    PROC rWireCut()
        VAR jointtarget jTepmCut{10};
        VAR speeddata vTempFast;
        VAR speeddata vTempSlow;
        vTempFast:=[nWireCutSpeed,500,nWireCutSpeed,100];
        vTempSlow:=[nWireCutSpeed/3,500,nWireCutSpeed/3,100];
        PulseDO\PLength:=nInchingTime,soAwManFeedFwd;
        Reset do09_Wire_Cutter_Close;
        Set do10_Wire_Cutter_Open;
        !      WaitTime 2.25;
        jWireCut4.robax:=[90,90,-50,0,0,0];
        MoveAbsJ jWireCut4\NoEOffs,vTempFast,z100,tWeld1;
        MoveAbsJ jWireCut3\NoEOffs,vTempFast,z100,tWeld1;
        MoveAbsJ jWireCut2\NoEOffs,vTempFast,z100,tWeld1;
        MoveAbsJ jWireCut1\NoEOffs,vTempFast,z10,tWeld1;
        WaitRob\ZeroSpeed;
        WaitTime 0.3;
        MoveAbsJ jWireCut0\NoEOffs,vTempSlow,z0,tWeld1;
        IF bWireCutSync=TRUE WaitSyncTask Wait{90},taskGroup12;
        WaitRob\ZeroSpeed;
        WaitTime 0.5;
        Reset do10_Wire_Cutter_Open;
        PulseDO\PLength:=1,do09_Wire_Cutter_Close;
        WaitTime 0.5;
        PulseDO\PLength:=1,do10_Wire_Cutter_Open;
        WaitTime 1;
        MoveAbsJ jWireCut1\NoEOffs,vTempSlow,z100,tWeld1;
        WaitRob\ZeroSpeed;
        MoveAbsJ jWireCut2\NoEOffs,vTempFast,z100,tWeld1;
        MoveAbsJ jWireCut3\NoEOffs,vTempFast,z100,tWeld1;
        MoveAbsJ jWireCut4\NoEOffs,vTempFast,z100,tWeld1;
        WaitRob\ZeroSpeed;
        Reset do10_Wire_Cutter_Open;
        stReact{1}:="WireCutOk";
        WaitUntil stCommand="";
        stReact{1}:="Ready";
        WaitUntil stReact=["Ready","Ready","Ready"];
        RETURN ;
    ENDPROC

    PROC rWireCutMove()
        VAR jointtarget jTepmCut{10};
        VAR speeddata vTempFast;
        VAR speeddata vTempSlow;
        vTempFast:=[nWireCutSpeed,500,nWireCutSpeed,100];
        vTempSlow:=[nWireCutSpeed/3,500,nWireCutSpeed/3,100];
        PulseDO\PLength:=nInchingTime,soAwManFeedFwd;
        Reset do09_Wire_Cutter_Close;
        Set do10_Wire_Cutter_Open;
        !      WaitTime 2.25;
        MoveAbsJ jWireCut3\NoEOffs,vTempFast,z100,tWeld1;
        MoveAbsJ jWireCut2\NoEOffs,vTempFast,z100,tWeld1;
        MoveAbsJ jWireCut1\NoEOffs,vTempFast,z10,tWeld1;
        WaitRob\ZeroSpeed;
        WaitTime 0.3;
        MoveAbsJ jWireCut0\NoEOffs,vTempSlow,z0,tWeld1;
        IF bWireCutSync=TRUE WaitSyncTask Wait{90},taskGroup12;
        WaitRob\ZeroSpeed;
        WaitTime 0.5;
        Reset do10_Wire_Cutter_Open;
        PulseDO\PLength:=1,do09_Wire_Cutter_Close;
        WaitTime 0.5;
        PulseDO\PLength:=1,do10_Wire_Cutter_Open;
        WaitTime 1;
        MoveAbsJ jWireCut1\NoEOffs,vTempSlow,z100,tWeld1;
        WaitRob\ZeroSpeed;
        MoveAbsJ jWireCut2\NoEOffs,vTempFast,z100,tWeld1;
        IF bWirecut=[FALSE,TRUE,FALSE] THEN
            MoveAbsJ jWireCut3\NoEOffs,vTempFast,z100,tWeld1;
            jWireCut4.robax:=[40,90,-90,0,0,0];
            MoveAbsJ jWireCut4\NoEOffs,vTempFast,z100,tWeld1;
        ENDIF
        WaitRob\ZeroSpeed;
        Reset do10_Wire_Cutter_Open;
        stReact{1}:="WireCutOk";
        WaitUntil stCommand="";
        stReact{1}:="Ready";
        WaitUntil stReact=["Ready","Ready","Ready"];
        RETURN ;
    ENDPROC

    PROC rWireCutShot()
        VAR jointtarget jTepmCut{10};
        VAR speeddata vTempFast;
        VAR speeddata vTempSlow;
        vTempFast:=[nWireCutSpeed,500,nWireCutSpeed,100];
        vTempSlow:=[nWireCutSpeed/3,500,nWireCutSpeed/3,100];
        PulseDO\PLength:=nInchingTime,soAwManFeedFwd;
        Reset do09_Wire_Cutter_Close;
        Set do10_Wire_Cutter_Open;
        WaitTime nInchingTime;
        MoveAbsJ jWireCut1\NoEOffs,vTempFast,z10,tWeld1;
        WaitRob\ZeroSpeed;
        WaitTime 0.3;
        MoveAbsJ jWireCut0\NoEOffs,vTempSlow,z0,tWeld1;
        IF bWireCutSync=TRUE WaitSyncTask Wait{90},taskGroup12;
        WaitRob\ZeroSpeed;
        WaitTime 0.5;
        Reset do10_Wire_Cutter_Open;
        PulseDO\PLength:=1,do09_Wire_Cutter_Close;
        WaitTime 0.5;
        PulseDO\PLength:=1,do10_Wire_Cutter_Open;
        WaitTime 1;
        MoveAbsJ jWireCut1\NoEOffs,vTempSlow,z100,tWeld1;
        WaitRob\ZeroSpeed;
        MoveAbsJ jWireCut2\NoEOffs,vTempFast,z100,tWeld1;
        WaitRob\ZeroSpeed;
        Reset do10_Wire_Cutter_Open;
        stReact{1}:="WireCutOk";
        WaitUntil stCommand="";
        stReact{1}:="Ready";
        WaitUntil stReact=["Ready","Ready","Ready"];
        RETURN ;
    ENDPROC

    PROC rTrapNoWeldMove()
        VAR num i;
        VAR targetdata WeldsTemp;
        VAR robtarget pWeldTemp;
        VAR num nTempMmps;
        VAR speeddata vWeldTemp;
        IDelete inumMoveG_PosHold;
        StopMove;
        !        ClearPath;
        !        StorePath;

        i:=nRunningStep{1};
        nTempMmps:=Welds1{i}.cpm/6;
        vWeldTemp:=[nTempMmps,200,200,200];

        pWeldTemp:=CRobT(\taskname:="T_ROB1"\Tool:=tWeld1\WObj:=wobjWeldLine1);
        StartMove;
        ConfL\Off;
        WHILE (so_MoveG_PosHold=1) DO
            nTrapCheck_1:=2;
            MoveL Offs(pWeldTemp,0,0,0),vWeldTemp,fine,tWeld1\WObj:=wobjWeldLine1;
            MoveL Offs(pWeldTemp,0,0,0),vWeldTemp,fine,tWeld1\WObj:=wobjWeldLine1;
        ENDWHILE
        ConfL\On;
        !        RestoPath;
    ENDPROC

    PROC rCorrSearchStartEnd()
        VAR num TempHeight;
        VAR num TempBreadth;
        VAR num Temp_X;
        VAR num Temp_Y;
        VAR num nHeightBuffer;
        VAR num n_X;
        VAR num n_Y;
        VAR num n_Z;
        VAR num n_Ret_X;
        VAR num n_Ret_Y;
        VAR num n_Ret_Z;
        VAR robtarget pTemp;
        VAR robtarget pCorrTemp_Start{2};
        VAR jointtarget jCorrTemp_Start{2};
        VAR robtarget pCorrTemp_End{2};
        VAR jointtarget jCorrTemp_End{2};

        RetryDepthData:=[10,10,10];
        IDelete iErrorDuringEntry;
        CONNECT iErrorDuringEntry WITH trapErrorDuringEntry;
        ISignalDO intTouch_1,1,iErrorDuringEntry;
        ISleep iErrorDuringEntry;

        bInstalldir:=bRobSwap;
        IF bRobSwap=FALSE THEN
            edgestartBuffer1:=edgeStart{1};
            edgeEndBuffer1:=edgeEnd{1};
        ELSE
            edgestartBuffer1:=edgeStart{2};
            edgeEndBuffer1:=edgeEnd{2};
        ENDIF
        WaitRob\ZeroSpeed;
        WaitSyncTask Wait{20},taskGroup123;

        WaitUntil bGanTry_Last_pos=TRUE;
        !        IF pi29_NextCmd=1 nTouchRetryCount{1}:=0;

        nCorrFailOffs_Z:=10*nEntryRetryCount{1};
        IF bRobSwap=TRUE nCorrFailOffs_Y:=(10*nEntryRetryCount{1});
        IF bRobSwap=FALSE nCorrFailOffs_Y:=(10*nEntryRetryCount{1});


        TEST nMacro001{1}
        CASE 0,1,2,3,4,5,8:
            IF edgeEndBuffer1.Breadth<edgeEndBuffer1.Height THEN
                ! Setting Conditions
                IF nMacro001{1}=0 OR nMacro001{1}=1 OR nMacro001{1}=2 OR nMacro001{1}=5 n_X:=-15;
                IF nMacro001{1}=3 OR nMacro001{1}=4 OR nMacro001{1}=8 n_X:=0;
                !                n_Y:=TouchLimit(corrEnd{nMacro001{1}+1}.Y_StartOffset+nEndThick,edgeEndBuffer1.Breadth)+nCorrFailOffs_Y;
                n_Y:=corrEnd{nMacro001{1}+1}.Y_StartOffset+nEndThick+nCorrFailOffs_Y;
                n_Ret_Y:=TouchLimit(corrEnd{nMacro001{1}+1}.Y_ReturnLength,edgeEndBuffer1.Breadth);
                n_Ret_Z:=TouchLimit(corrEnd{nMacro001{1}+1}.Z_ReturnLength,edgeEndBuffer1.Height);
                n_Z:=TouchLimit(corrEnd{nMacro001{1}+1}.Z_StartOffset,edgeEndBuffer1.Height)+nCorrFailOffs_Z;

                ! Touch Entry Location================================================================
                IWatch iErrorDuringEntry;

                rCheckWelder;

                rMoveCorrConnect n_X,n_Y,n_Z,0,0,0,nHeightBuffer,bEnd,bInstalldir\LIN;
                Reset soLn1Touch;
                IDelete iErrorDuringEntry;

                !                IF bTouchWorkCount{3}=TRUE GOTO TouchComplete_End_Y;
                WaitTime 0;
                !                 rCheckTouchAtStart;
                !=====================================================================================
                ! edge_Y
                IF bTouchWorkCount{1}=FALSE THEN
                    rCorrSearchWeldLineEdgeY n_X,n_Y,n_Z,corrEnd{nMacro001{1}+1}.Y_Depth+nCorrFailOffs_Y+nEndThick,n_Ret_Y,bEnd,bInstalldir,"End_Y";
                    bTouchWorkCount{1}:=TRUE;
                    nTouchRetryCount{1}:=0;
                ENDIF

                ! edge_Z
                IF bTouchWorkCount{2}=FALSE THEN
                    !                 Setting Conditions
                    n_Y:=n_Ret_Y;
                    n_Ret_Z:=TouchLimit(corrEnd{nMacro001{1}+1}.Z_ReturnLength,edgeEndBuffer1.Height);

                    rCorrSearchWeldLineEdgeZ n_X,n_Y,n_Z,corrEnd{nMacro001{1}+1}.Z_Depth+nCorrFailOffs_Z,n_Ret_Z,bEnd,bInstalldir,"End_Z";
                    bTouchWorkCount{2}:=TRUE;
                    nTouchRetryCount{1}:=0;
                ENDIF

                ! Setting Conditions
                n_Z:=n_Ret_Z;
                rMoveCorrConnect n_X,n_Y,n_Z,0,0,0,nHeightBuffer,bEnd,bInstalldir;

                IF nMacro001{1}=3 OR nMacro001{1}=4 OR nMacro001{1}=8 GOTO TouchComplete_End_Y;
                IF nMacro001{1}=2 OR nMacro001{1}=5 THEN
                    IF nMacro001{1}=5 n_Z:=edgeEndBuffer1.HoleSize+1;
                ELSE
                    ! Setting Conditions
                    n_X:=corrEnd{nMacro001{1}+1}.X_StartOffset;
                    rMoveCorrConnect n_X,n_Y,n_Z,0,0,0,nHeightBuffer,bEnd,bInstalldir;
                    ! Setting Conditions
                    n_Y:=-5;
                    rMoveCorrConnect n_X,n_Y,n_Z,0,0,0,nHeightBuffer,bEnd,bInstalldir;

                ENDIF

                ! edge_X
                IF bTouchWorkCount{3}=FALSE THEN
                    rCorrSearchWeldLineEdgeX n_X,n_Y,n_Z,corrEnd{nMacro001{1}+1}.X_Depth,corrEnd{nMacro001{1}+1}.X_ReturnLength,bEnd,bInstalldir,"End_X";
                    bTouchWorkCount{3}:=TRUE;
                    nTouchRetryCount{1}:=0;
                ENDIF
                ! Setting Conditions
                n_X:=corrEnd{nMacro001{1}+1}.X_ReturnLength;
                rMoveCorrConnect n_X,n_Y,n_Z,0,corrEnd{nMacro001{1}+1}.RY_Torch,0,nHeightBuffer,bEnd,bInstalldir;
                ! Labal
                TouchComplete_End_Y:
                ! Setting Conditions
                n_Y:=n_Ret_Y;
                rMoveCorrConnect n_X,n_Y,n_Z,0,corrEnd{nMacro001{1}+1}.RY_Torch+n_Angle,0,nHeightBuffer,bEnd,bInstalldir;

            ELSE

                ! Setting Conditions
                IF nMacro001{1}=0 OR nMacro001{1}=1 OR nMacro001{1}=2 OR nMacro001{1}=5 n_X:=-15;
                IF nMacro001{1}=3 OR nMacro001{1}=4 OR nMacro001{1}=8 n_X:=0;
                n_Y:=TouchLimit(corrEnd{nMacro001{1}+1}.Y_StartOffset+nEndThick,edgeEndBuffer1.Breadth)+nCorrFailOffs_Y;
                n_Ret_Y:=TouchLimit(corrEnd{nMacro001{1}+1}.Y_ReturnLength,edgeEndBuffer1.Breadth);
                n_Ret_Z:=TouchLimit(corrEnd{nMacro001{1}+1}.Z_ReturnLength,edgeEndBuffer1.Height);
                n_Z:=TouchLimit(corrEnd{nMacro001{1}+1}.Z_StartOffset,edgeEndBuffer1.Height)+nCorrFailOffs_Z;

                IWatch iErrorDuringEntry;

                rCheckWelder;

                rMoveCorrConnect n_X,n_Y,n_Z,0,0,0,nHeightBuffer,bEnd,bInstalldir\LIN;
                Reset soLn1Touch;
                IDelete iErrorDuringEntry;

                !                IF bTouchWorkCount{3}=TRUE GOTO TouchComplete_End_Z;
                WaitTime 0;
                !    rCheckTouchAtStart;

                ! edge_Z
                IF bTouchWorkCount{1}=FALSE THEN
                    rCorrSearchWeldLineEdgeZ n_X,n_Y,n_Z,corrEnd{nMacro001{1}+1}.Z_Depth+nCorrFailOffs_Z,n_Ret_Z,bEnd,bInstalldir,"End_Z";
                    bTouchWorkCount{1}:=TRUE;
                    nTouchRetryCount{1}:=0;
                ENDIF

                ! edge_Y
                IF bTouchWorkCount{2}=FALSE THEN
                    ! Setting Conditions
                    n_Ret_Y:=TouchLimit(corrEnd{nMacro001{1}+1}.Y_ReturnLength,edgeEndBuffer1.Breadth);
                    n_Z:=n_Ret_Z;
                    rCorrSearchWeldLineEdgeY n_X,n_Y,n_Z,corrEnd{nMacro001{1}+1}.Y_Depth+nCorrFailOffs_Y+nEndThick,n_Ret_Y,bEnd,bInstalldir,"End_Y";
                    bTouchWorkCount{2}:=TRUE;
                    nTouchRetryCount{1}:=0;
                ENDIF

                ! Setting Conditions
                n_Y:=n_Ret_Y;
                rMoveCorrConnect n_X,n_Y,n_Z,0,0,0,nHeightBuffer,bEnd,bInstalldir;

                IF nMacro001{1}=3 OR nMacro001{1}=4 OR nMacro001{1}=8 GOTO TouchComplete_End_Z;
                IF nMacro001{1}=2 OR nMacro001{1}=5 THEN
                    IF nMacro001{1}=5 n_Z:=edgeEndBuffer1.HoleSize+1;
                ELSE

                    ! Setting Conditions
                    n_X:=corrEnd{nMacro001{1}+1}.X_StartOffset;
                    rMoveCorrConnect n_X,n_Y,n_Z,0,0,0,nHeightBuffer,bEnd,bInstalldir;
                    ! Setting Conditions
                    n_Y:=-5;
                    rMoveCorrConnect n_X,n_Y,n_Z,0,0,0,nHeightBuffer,bEnd,bInstalldir;

                ENDIF

                ! edge_X
                IF bTouchWorkCount{3}=FALSE THEN
                    rCorrSearchWeldLineEdgeX n_X,n_Y,n_Z,corrEnd{nMacro001{1}+1}.X_Depth,corrEnd{nMacro001{1}+1}.X_ReturnLength,bEnd,bInstalldir,"End_X";
                    bTouchWorkCount{3}:=TRUE;
                    nTouchRetryCount{1}:=0;
                ENDIF

                ! Setting Conditions
                n_X:=corrEnd{nMacro001{1}+1}.X_ReturnLength;
                rMoveCorrConnect n_X,n_Y,n_Z,0,corrEnd{nMacro001{1}+1}.RY_Torch,0,nHeightBuffer,bEnd,bInstalldir;
                ! Labal
                TouchComplete_End_Z:
                ! Setting Conditions
                n_Y:=n_Ret_Y;
                rMoveCorrConnect n_X,n_Y,n_Z,0,corrEnd{nMacro001{1}+1}.RY_Torch+n_Angle,0,nHeightBuffer,bEnd,bInstalldir;
            ENDIF
            IF nMacro001{1}=3 OR nMacro001{1}=4 OR nMacro001{1}=8 THEN
                !   IF bEndSearchComplete=FALSE pCorredSplitPos:=ConvertPosWeldLineToFloor(pSearchStart,nWeldLineLength+nCorrX_Store_End,nCorrY_Store_End,nCorrZ_Store_End);
            ENDIF
        CASE 9:
            !   pCorredEndPos:=pCorredSplitPos;
        DEFAULT:
            Stop;
            Stop;
            ExitCycle;
        ENDTEST

        !        IF abs(pCheckBuffer{2}.trans.x-pCheckBuffer{3}.trans.x)<5 rTouchErrorHandling 13;
        !        IF abs(pCheckBuffer{2}.trans.Y-pCheckBuffer{3}.trans.Y)<5 rTouchErrorHandling 13;
        !        IF abs(pCheckBuffer{2}.trans.Z-pCheckBuffer{3}.trans.Z)<5 rTouchErrorHandling 13;

        bTouch_last_R1_Comp:=TRUE;
        bTouch_First_R1_Comp:=FALSE;
        pCorrTemp_End{1}:=CRobT(\TaskName:="T_ROB1"\Tool:=tWeld1\WObj:=wobjWeldLine1);
        pCorrTemp_End{1}.trans:=[nWeldLineLength_R1+nCorrX_Store_End{1},nCorrY_Store_End{1},nCorrZ_Store_End{1}];
        jCorrTemp_End{1}:=CalcJointT(pCorrTemp_End{1},tWeld1\WObj:=wobjWeldLine1);
        pCorrT_ROB1_End:=CalcRobT(jCorrTemp_End{1},Tool:=tWeld1\WObj:=wobjRotCtr1);
        WaitUntil bGanTry_First_pos=TRUE AND bTouch_last_R2_Comp=TRUE;

        !!! Start correctioning from start edge !!!
        TEST nMacro010{1}
        CASE 0,1,2,3,4,5:
            IF edgestartBuffer1.Breadth<edgestartBuffer1.Height THEN

                ! Setting Conditions
                IF nMacro010{1}=0 OR nMacro010{1}=1 OR nMacro010{1}=2 OR nMacro010{1}=5 n_X:=-15;
                IF nMacro010{1}=3 OR nMacro010{1}=4 OR nMacro010{1}=8 n_X:=0;
                !                n_Y:=TouchLimit(corrStart{nMacro010{1}+1}.Y_StartOffset+nStartThick,edgeStartBuffer1.Breadth)+nCorrFailOffs_Y;
                n_Y:=corrStart{nMacro010{1}+1}.Y_StartOffset+nStartThick+nCorrFailOffs_Y;
                n_Ret_Y:=TouchLimit(corrStart{nMacro010{1}+1}.Y_ReturnLength,edgestartBuffer1.Breadth);
                n_Z:=TouchLimit(corrStart{nMacro010{1}+1}.Z_StartOffset,edgestartBuffer1.Height)+nCorrFailOffs_Z;
                n_Ret_Z:=TouchLimit(corrStart{nMacro010{1}+1}.Z_ReturnLength,edgestartBuffer1.Height);

                ! edge_Y
                rMoveCorrConnect n_X,n_Y,n_Z,0,corrStart{nMacro010{1}+1}.RY_Torch+n_Angle,0,nHeightBuffer,bStart,bInstalldir\LIN;
                !    rCheckTouchAtStart;

                IF bTouchWorkCount{4}=FALSE THEN
                    rCorrSearchWeldLineEdgeY n_X,n_Y,n_Z,corrStart{nMacro010{1}+1}.Y_Depth+nCorrFailOffs_Y+nStartThick,n_Ret_Y,bStart,bInstalldir,"Start_Y";
                    bTouchWorkCount{4}:=TRUE;
                    nTouchRetryCount{1}:=0;
                ENDIF

                ! edge_Z
                IF bTouchWorkCount{5}=FALSE THEN
                    ! Setting Conditions
                    n_Y:=n_Ret_Y;
                    n_Ret_Z:=TouchLimit(corrStart{nMacro010{1}+1}.Z_ReturnLength,edgestartBuffer1.Height);
                    rCorrSearchWeldLineEdgeZ n_X,n_Y,n_Z,corrStart{nMacro010{1}+1}.Z_Depth+nCorrFailOffs_Z,n_Ret_Z,bStart,bInstalldir,"Start_Z";
                    bTouchWorkCount{5}:=TRUE;
                    nTouchRetryCount{1}:=0;
                ENDIF

                ! Setting Conditions
                n_Z:=n_Ret_Z;
                rMoveCorrConnect n_X,n_Y,n_Z,0,0,0,nHeightBuffer,bStart,bInstalldir;

                IF nMacro010{1}=3 OR nMacro010{1}=4 OR nMacro010{1}=8 GOTO TouchComplete_Start_Y;
                IF nMacro010{1}=2 OR nMacro010{1}=5 THEN
                    IF nMacro010{1}=5 n_Z:=edgestartBuffer1.HoleSize+1;
                ELSE

                    ! Setting Conditions
                    n_X:=corrStart{nMacro010{1}+1}.X_StartOffset;
                    rMoveCorrConnect n_X,n_Y,n_Z,0,0,0,nHeightBuffer,bStart,bInstalldir;
                    ! Setting Conditions
                    n_Y:=-5;
                    rMoveCorrConnect n_X,n_Y,n_Z,0,0,0,nHeightBuffer,bStart,bInstalldir;
                ENDIF
                !    ENDIF

                ! edge_X
                IF bTouchWorkCount{6}=FALSE THEN
                    rCorrSearchWeldLineEdgeX n_X,n_Y,n_Z,corrStart{nMacro010{1}+1}.X_Depth,corrStart{nMacro010{1}+1}.X_ReturnLength,bStart,bInstalldir,"Start_X";
                    bTouchWorkCount{6}:=TRUE;
                    nTouchRetryCount{1}:=0;
                ENDIF
                ! Setting Conditions
                n_X:=corrStart{nMacro010{1}+1}.X_ReturnLength;
                rMoveCorrConnect n_X,n_Y,n_Z,0,corrStart{nMacro010{1}+1}.RY_Torch,0,nHeightBuffer,bStart,bInstalldir;
                ! Labal
                TouchComplete_Start_Y:
            ELSE

                ! Setting Conditions
                IF nMacro010{1}=0 OR nMacro010{1}=1 OR nMacro010{1}=2 OR nMacro010{1}=5 n_X:=-15;
                IF nMacro010{1}=3 OR nMacro010{1}=4 OR nMacro010{1}=8 n_X:=0;
                n_Y:=TouchLimit(corrStart{nMacro010{1}+1}.Y_StartOffset+nStartThick,edgestartBuffer1.Breadth)+nCorrFailOffs_Y;
                n_Ret_Y:=TouchLimit(corrStart{nMacro010{1}+1}.Y_ReturnLength,edgestartBuffer1.Breadth);
                n_Ret_Z:=TouchLimit(corrStart{nMacro010{1}+1}.Z_ReturnLength,edgestartBuffer1.Height);
                n_Z:=TouchLimit(corrStart{nMacro010{1}+1}.Z_StartOffset,edgestartBuffer1.Height)+nCorrFailOffs_Z;

                rMoveCorrConnect n_X,n_Y,n_Z,0,corrStart{nMacro010{1}+1}.RY_Torch+n_Angle,0,nHeightBuffer,bStart,bInstalldir\LIN;
                ! rCheckTouchAtStart;


                ! edge_Z
                IF bTouchWorkCount{4}=FALSE THEN
                    rCorrSearchWeldLineEdgeZ n_X,n_Y,n_Z,corrStart{nMacro010{1}+1}.Z_Depth+nCorrFailOffs_Z,n_Ret_Z,bStart,bInstalldir,"Start_Z";
                    bTouchWorkCount{4}:=TRUE;
                    nTouchRetryCount{1}:=0;
                ENDIF
                ! Setting Conditions


                ! edge_Y
                IF bTouchWorkCount{5}=FALSE THEN
                    ! Setting Conditions
                    n_Ret_Y:=TouchLimit(corrStart{nMacro010{1}+1}.Y_ReturnLength,edgestartBuffer1.Breadth);
                    n_Z:=n_Ret_Z;
                    rCorrSearchWeldLineEdgeY n_X,n_Y,n_Z,corrStart{nMacro010{1}+1}.Y_Depth+nCorrFailOffs_Y+nStartThick,n_Ret_Y,bStart,bInstalldir,"Start_Y";
                    bTouchWorkCount{5}:=TRUE;
                    nTouchRetryCount{1}:=0;
                ENDIF

                ! Setting Conditions
                n_Y:=n_Ret_Y;
                rMoveCorrConnect n_X,n_Y,n_Z,0,0,0,nHeightBuffer,bStart,bInstalldir;

                IF nMacro010{1}=3 OR nMacro010{1}=4 OR nMacro010{1}=8 GOTO TouchComplete_Start_Z;
                IF nMacro010{1}=2 OR nMacro010{1}=5 THEN
                    IF nMacro010{1}=5 n_Z:=edgestartBuffer1.HoleSize+1;
                ELSE
                    !    IF bTouchWorkCount{6}=FALSE THEN
                    ! Setting Conditions
                    n_X:=corrStart{nMacro010{1}+1}.X_StartOffset;
                    rMoveCorrConnect n_X,n_Y,n_Z,0,0,0,nHeightBuffer,bStart,bInstalldir;
                    ! Setting Conditions
                    n_Y:=-5;
                    rMoveCorrConnect n_X,n_Y,n_Z,0,0,0,nHeightBuffer,bStart,bInstalldir;
                ENDIF
                ! ENDIF

                ! edge_X
                IF bTouchWorkCount{6}=FALSE THEN
                    rCorrSearchWeldLineEdgeX n_X,n_Y,n_Z,corrStart{nMacro010{1}+1}.X_Depth,corrStart{nMacro010{1}+1}.X_ReturnLength,bStart,bInstalldir,"Start_X";
                    bTouchWorkCount{6}:=TRUE;
                    nTouchRetryCount{1}:=0;
                ENDIF
                ! Setting Conditions
                n_X:=corrStart{nMacro010{1}+1}.X_ReturnLength;
                rMoveCorrConnect n_X,n_Y,n_Z,0,corrStart{nMacro010{1}+1}.RY_Torch,0,nHeightBuffer,bStart,bInstalldir;

                ! Labal
                TouchComplete_Start_Z:
            ENDIF

        DEFAULT:
            Stop;
            Stop;
            ExitCycle;
        ENDTEST

        pTemp:=CRobT(\TaskName:="T_ROB1"\Tool:=tWeld1\WObj:=wobjWeldLine1);
        WaitRob\ZeroSpeed;
        MoveL RelTool(pTemp,0,0,-15),vTargetSpeed,zTargetZone,tWeld1\WObj:=wobjWeldLine1;

        bTouch_First_R1_Comp:=TRUE;
        bTouch_last_R1_Comp:=TRUE;

        WaitUntil bTouch_First_R2_Comp=TRUE;

        pCorrTemp_Start{1}:=CRobT(\TaskName:="T_ROB1"\Tool:=tWeld1\WObj:=wobjWeldLine1);
        pCorrTemp_Start{1}.trans:=[nCorrX_Store_Start{1},nCorrY_Store_Start{1},nCorrZ_Store_Start{1}];
        jCorrTemp_Start{1}:=CalcJointT(pCorrTemp_Start{1},tWeld1\WObj:=wobjWeldLine1);
        pCorrT_ROB1_Start:=CalcRobT(jCorrTemp_Start{1},Tool:=tWeld1\WObj:=wobjRotCtr1);








        stReact{1}:="CorrSearchOK";
        WaitUntil stCommand="";
        stReact{1}:="Ready";
        nCorrFailOffs_Y:=0;
        nCorrFailOffs_Z:=0;
        nCorrX_Store_Start{1}:=0;
        nCorrY_Store_Start{1}:=0;
        nCorrZ_Store_Start{1}:=0;
        nCorrX_Store_End{1}:=0;
        nCorrY_Store_End{1}:=0;
        nCorrZ_Store_End{1}:=0;
    ENDPROC

    PROC rMoveCorrConnect(num X,num Y,num Z,num Rx,num Ry,num Rz,num EAX_D,bool isStartPos,bool CCW,\switch LIN)
        VAR robtarget pTempConnect;
        VAR num nCorrX_Store;
        VAR num nCorrY_Store;
        VAR num nCorrZ_Store;

        IF (isStartPos=bStart) THEN
            nCorrX_Store:=nCorrX_Store_Start{1};
            nCorrY_Store:=nCorrY_Store_Start{1};
            nCorrZ_Store:=nCorrZ_Store_Start{1};
        ELSE
            nCorrX_Store:=nCorrX_Store_End{1};
            nCorrY_Store:=nCorrY_Store_End{1};
            nCorrZ_Store:=nCorrZ_Store_End{1};
        ENDIF


        pTempConnect:=pNull;
        pTempConnect.robconf:=[0,0,0,1];

        IF isStartPos=bStart THEN
            IF CCW=FALSE THEN
                pTempConnect.trans:=[nCorrX_Store+(-1*X),nCorrY_Store+(Y),nCorrZ_Store+(Z)];
                pTempConnect.rot:=[0.5,0.5,-0.5,0.5];
                pTempConnect:=RelTool(pTempConnect,0,0,0\Rx:=-1*macroStartBuffer1{1}.TravelAngle\Ry:=-1*macroStartBuffer1{1}.WorkingAngle+nBreakPoint{1});
            ELSE
                pTempConnect.trans:=[nCorrX_Store+(-1*X),nCorrY_Store+(-1*Y),nCorrZ_Store+(Z)];
                pTempConnect.rot:=[0.5,-0.5,-0.5,-0.5];
                pTempConnect:=RelTool(pTempConnect,0,0,0\Rx:=macroStartBuffer1{1}.TravelAngle\Ry:=-1*macroStartBuffer1{1}.WorkingAngle+nBreakPoint{1});

            ENDIF
        ELSEIF isStartPos=bEnd THEN
            IF CCW=FALSE THEN
                pTempConnect.trans:=[nWeldLineLength_R1+nCorrX_Store+(X),nCorrY_Store+(Y),nCorrZ_Store+(Z)];
                pTempConnect.rot:=[0.5,0.5,-0.5,0.5];
                pTempConnect:=RelTool(pTempConnect,0,0,0\Rx:=-1*macroEndBuffer1{nMotionEndStepLast{1}}.TravelAngle\Ry:=-1*macroEndBuffer1{nMotionEndStepLast{1}}.WorkingAngle+nBreakPoint{1});
            ELSE
                pTempConnect.trans:=[nWeldLineLength_R1+nCorrX_Store+(X),nCorrY_Store+(-1*Y),nCorrZ_Store+(Z)];
                pTempConnect.rot:=[0.5,-0.5,-0.5,-0.5];
                pTempConnect:=RelTool(pTempConnect,0,0,0\Rx:=macroEndBuffer1{nMotionEndStepLast{1}}.TravelAngle\Ry:=-1*macroEndBuffer1{nMotionEndStepLast{1}}.WorkingAngle+nBreakPoint{1});
            ENDIF
        ENDIF

        IF Present(LIN)=FALSE THEN
            MoveJ pTempConnect,v300,fine,tWeld1\WObj:=wobjWeldLine1;
        ELSE
            MoveL pTempConnect,v300,fine,tWeld1\WObj:=wobjWeldLine1;
        ENDIF

        RETURN ;
    ENDPROC

    PROC rCorrSearchWeldLineEdgeX(num X,num Y,num Z,num Depth,num RetX,bool isStartPos,bool CCW,string dirErrorCheck)
        VAR num nCorrX_Store;
        VAR num nCorrY_Store;
        VAR num nCorrZ_Store;

        WaitUntil bRobSwap=CCW;
        IF (isStartPos=bStart) THEN
            nCorrX_Store:=nCorrX_Store_Start{1};
            nCorrY_Store:=nCorrY_Store_Start{1};
            nCorrZ_Store:=nCorrZ_Store_Start{1};
        ELSE
            nCorrX_Store:=nCorrX_Store_End{1};
            nCorrY_Store:=nCorrY_Store_End{1};
            nCorrZ_Store:=nCorrZ_Store_End{1};
        ENDIF

        TouchErrorDirSub:=dirErrorCheck;
        IF TouchErrorDirMain=dirErrorCheck AND 0<nTouchRetryCount{1} THEN
            IF (isStartPos=bEnd AND (nMacro001{1}=2 OR nMacro001{1}=5)) OR (isStartPos=bStart AND (nMacro010{1}=2 OR nMacro010{1}=5)) THEN
                Depth:=Depth+((RetryDepthData{1}*(-1))*nTouchRetryCount{1});
            ELSE
                Depth:=Depth+(RetryDepthData{1}*nTouchRetryCount{1});
            ENDIF
        ENDIF
        !!! Search weld X edge !!!
        WaitUntil bRobSwap=CCW;
        IF (isStartPos=bStart) THEN
            pSearchStart.rot:=Welds1{1}.position.rot;
            IF (CCW=FALSE) pSearchStart.trans:=[nCorrX_Store+(-1*X),nCorrY_Store+(Y),nCorrZ_Store+(Z)];
            IF (CCW=TRUE) pSearchStart.trans:=[nCorrX_Store+(-1*X),nCorrY_Store+(-1*Y),nCorrZ_Store+(Z)];
        ELSEIF (isStartPos=bEnd) THEN
            pSearchStart.rot:=Welds1{nMotionStepCount{1}}.position.rot;
            IF (CCW=FALSE) pSearchStart.trans:=[nWeldLineLength_R1+nCorrX_Store+(X),nCorrY_Store+(Y),nCorrZ_Store+(Z)];
            IF (CCW=TRUE) pSearchStart.trans:=[nWeldLineLength_R1+nCorrX_Store+(X),nCorrY_Store+(-1*Y),nCorrZ_Store+(Z)];
        ENDIF

        pSearchStart.robconf.cfx:=1;
        pSearchStart.extax:=[9e9,9e9,9e9,9e9,9e9,9e9];

        pSearchEnd:=pSearchStart;
        IF (isStartPos=bStart) pSearchEnd.trans.x:=pSearchStart.trans.x+Depth;
        IF (isStartPos=bEnd) pSearchEnd.trans.x:=pSearchStart.trans.x-Depth;

        rCorrSearchByWire pSearchStart,pSearchEnd\X;

        !        pCheckBuffer{1}.trans:=pCorredPosBuffer;

        IF (isStartPos=bStart) nCorrX_Store:=pCorredPosBuffer.x;
        IF (isStartPos=bEnd) nCorrX_Store:=pCorredPosBuffer.x-nWeldLineLength_R1;

        IF (isStartPos=bStart) THEN
            nCorrX_Store_Start{1}:=nCorrX_Store;
            nCorrY_Store_Start{1}:=nCorrY_Store;
            nCorrZ_Store_Start{1}:=nCorrZ_Store;
        ELSE
            nCorrX_Store_End{1}:=nCorrX_Store;
            nCorrY_Store_End{1}:=nCorrY_Store;
            nCorrZ_Store_End{1}:=nCorrZ_Store;
        ENDIF

        rMoveCorrConnect RetX,Y,Z,0,0,0,pSearchStart.extax.eax_d,isStartPos,CCW;
        nTouchRetryCount{1}:=0;
        TouchErrorDirMain:="Ready";

        RETURN ;
    ENDPROC

    PROC rCorrSearchWeldLineEdgeY(num X,num Y,num Z,num Depth,num RetY,bool isStartPos,bool CCW,string dirErrorCheck)
        VAR num nCorrX_Store;
        VAR num nCorrY_Store;
        VAR num nCorrZ_Store;
        WaitUntil bRobSwap=CCW;
        IF (isStartPos=bStart) THEN
            nCorrX_Store:=nCorrX_Store_Start{1};
            nCorrY_Store:=nCorrY_Store_Start{1};
            nCorrZ_Store:=nCorrZ_Store_Start{1};
        ELSE
            nCorrX_Store:=nCorrX_Store_End{1};
            nCorrY_Store:=nCorrY_Store_End{1};
            nCorrZ_Store:=nCorrZ_Store_End{1};
        ENDIF

        TouchErrorDirSub:=dirErrorCheck;
        IF (TouchErrorDirMain=dirErrorCheck AND 0<nTouchRetryCount{1}) Depth:=Depth+(RetryDepthData{2}*nTouchRetryCount{1});

        !!! Search weld Y edge !!!
        WaitUntil bRobSwap=CCW;
        IF (isStartPos=bStart) THEN
            pSearchStart.rot:=Welds1{1}.position.rot;
            IF (CCW=FALSE) pSearchStart.trans:=[nCorrX_Store+(-1*X),nCorrY_Store+(Y),nCorrZ_Store+(Z)];
            IF (CCW=TRUE) pSearchStart.trans:=[nCorrX_Store+(-1*X),nCorrY_Store+(-1*Y),nCorrZ_Store+Z];
        ELSEIF (isStartPos=bEnd) THEN
            pSearchStart.rot:=Welds1{nMotionStepCount{1}}.position.rot;
            IF (CCW=FALSE) pSearchStart.trans:=[nWeldLineLength_R1+nCorrX_Store+(X),nCorrY_Store+(Y),nCorrZ_Store+(Z)];
            IF (CCW=TRUE) pSearchStart.trans:=[nWeldLineLength_R1+nCorrX_Store+(X),nCorrY_Store+(-1*Y),nCorrZ_Store+(Z)];
        ENDIF

        pSearchStart.robconf.cfx:=1;

        pSearchEnd:=pSearchStart;
        pSearchStart.extax:=[9e9,9e9,9e9,9e9,9e9,9e9];
        IF (CCW=FALSE) pSearchEnd.trans.y:=pSearchStart.trans.y-Depth;
        IF (CCW=TRUE) pSearchEnd.trans.y:=pSearchStart.trans.y+Depth;

        rCorrSearchByWire pSearchStart,pSearchEnd\Y;

        !        pCheckBuffer{2}.trans:=pCorredPosBuffer;

        nCorrY_Store:=pCorredPosBuffer.y;

        IF (isStartPos=bStart) THEN
            nCorrX_Store_Start{1}:=nCorrX_Store;
            nCorrY_Store_Start{1}:=nCorrY_Store;
            nCorrZ_Store_Start{1}:=nCorrZ_Store;
        ELSE
            nCorrX_Store_End{1}:=nCorrX_Store;
            nCorrY_Store_End{1}:=nCorrY_Store;
            nCorrZ_Store_End{1}:=nCorrZ_Store;
        ENDIF

        rMoveCorrConnect X,RetY,Z,0,0,0,pSearchStart.extax.eax_d,isStartPos,CCW;
        nTouchRetryCount{1}:=0;
        TouchErrorDirMain:="Ready";

        RETURN ;
    ENDPROC

    PROC rCorrSearchWeldLineEdgeZ(num X,num Y,num Z,num Depth,num RetZ,bool isStartPos,bool CCW,string dirErrorCheck)
        VAR num nCorrX_Store;
        VAR num nCorrY_Store;
        VAR num nCorrZ_Store;
        WaitUntil bRobSwap=CCW;
        IF (isStartPos=bStart) THEN
            nCorrX_Store:=nCorrX_Store_Start{1};
            nCorrY_Store:=nCorrY_Store_Start{1};
            nCorrZ_Store:=nCorrZ_Store_Start{1};
        ELSE
            nCorrX_Store:=nCorrX_Store_End{1};
            nCorrY_Store:=nCorrY_Store_End{1};
            nCorrZ_Store:=nCorrZ_Store_End{1};
        ENDIF
        TouchErrorDirSub:=dirErrorCheck;
        IF (TouchErrorDirMain=dirErrorCheck AND 0<nTouchRetryCount{1}) Depth:=Depth+(RetryDepthData{3}*nTouchRetryCount{1});
        !!! Search weld Z edge !!!
        WaitUntil bRobSwap=CCW;
        IF (isStartPos=bStart) THEN
            pSearchStart.rot:=Welds1{1}.position.rot;
            IF (CCW=FALSE) pSearchStart.trans:=[nCorrX_Store+(-1*X),nCorrY_Store+(Y),nCorrZ_Store+(Z)];
            IF (CCW=TRUE) pSearchStart.trans:=[nCorrX_Store+(-1*X),nCorrY_Store+(-1*Y),nCorrZ_Store+(Z)];
        ELSEIF (isStartPos=bEnd) THEN
            pSearchStart.rot:=Welds1{nMotionStepCount{1}}.position.rot;
            IF (CCW=FALSE) pSearchStart.trans:=[nWeldLineLength_R1+nCorrX_Store+(X),nCorrY_Store+(Y),nCorrZ_Store+(Z)];
            IF (CCW=TRUE) pSearchStart.trans:=[nWeldLineLength_R1+nCorrX_Store+(X),nCorrY_Store+(-1*Y),nCorrZ_Store+(Z)];
        ENDIF

        pSearchStart.robconf.cfx:=1;
        pSearchStart.extax:=[9e9,9e9,9e9,9e9,9e9,9e9];

        pSearchEnd:=pSearchStart;
        pSearchEnd.trans.z:=pSearchStart.trans.z-Depth;

        rCorrSearchByWire pSearchStart,pSearchEnd\Z;

        !        pCheckBuffer{3}.trans:=pCorredPosBuffer;

        nCorrZ_Store:=pCorredPosBuffer.z;

        IF (isStartPos=bStart) THEN
            nCorrX_Store_Start{1}:=nCorrX_Store;
            nCorrY_Store_Start{1}:=nCorrY_Store;
            nCorrZ_Store_Start{1}:=nCorrZ_Store;
        ELSE
            nCorrX_Store_End{1}:=nCorrX_Store;
            nCorrY_Store_End{1}:=nCorrY_Store;
            nCorrZ_Store_End{1}:=nCorrZ_Store;
        ENDIF

        rMoveCorrConnect X,Y,RetZ,0,0,0,pSearchStart.extax.eax_d,isStartPos,CCW;
        nTouchRetryCount{1}:=0;
        TouchErrorDirMain:="Ready";

        RETURN ;
    ENDPROC

    PROC rCorrSearchByWire(robtarget SearchStart,robtarget SearchEnd,\switch X\switch Y\switch Z)
        VAR robtarget pTemp:=[[0,0,0],[1,0,0,0],[0,0,0,0],[0,0,0,0,9E+09,9E+09]];

        MoveJ SearchStart,v100,fine,tWeld1\WObj:=wobjWeldLine1;

        rCheckWelder;
        SearchL\SStop,bWireTouch1,SearchStart,SearchEnd,v10,tWeld1\WObj:=wobjWeldLine1;

        Reset soLn1Touch;
        WaitTime 0;
        WaitUntil(siLn1TouchActive=0);
        pTemp:=CRobT(\taskname:="T_ROB1"\tool:=tWeld1\WObj:=wobjWeldLine1);
        pCorredPosBuffer:=pTemp.trans;
        RETURN ;
    ERROR

        TouchErrorDirMain:=TouchErrorDirSub;
        IDelete iMoveHome_RBT1;
        IF ERRNO=ERR_WHLSEARCH THEN

            rTouchErrorHandling 2;
        ELSEIF ERRNO=ERR_SIGSUPSEARCH THEN
            WaitTime 999;
            rTouchErrorHandling 3;
        ELSE
            rTouchErrorHandling 4;
        ENDIF
    ENDPROC

    PROC rZero()
        MoveAbsJ [[0,0,0,0,0,0],[9E+09,9E+09,9E+09,9E+09,9E+09,9E+09]]\NoEOffs,v200,fine,tool0;
    ENDPROC

    PROC rErrorDuringEntry()
        VAR robtarget pTemp;
        Reset soLn1Touch;
        IDelete iMoveHome_RBT1;
        StopMove;
        ClearPath;
        StartMove;

        pTemp:=CRobT(\TaskName:="T_ROB1"\Tool:=tWeld1\WObj:=wobjWeldLine1);
        MoveL RelTool(pTemp,0,0,-10),vTargetSpeed,fine,tWeld1\WObj:=wobjWeldLine1;

        stReact{1}:="Error_Arc_Touch";
        WaitSyncTask Wait{80},taskGroup123;

        WaitUntil stReact=["Error_Arc_Touch","Error_Arc_Touch","Error_Arc_Touch"];
        WaitSyncTask Wait{81},taskGroup123;

        WaitUntil stCommand="Error_Arc_Touch";
        stReact{1}:="";
        WaitUntil stCommand="";
        WaitSyncTask Wait{82},taskGroup123;

        !        WaitSyncTask Wait{81},taskGroup123;

        ExitCycle;
    ENDPROC

    PROC rArcError()
        VAR robtarget pTemp;
        TPWrite "TROB1_ArcError";
        bArc_On{1}:=FALSE;
        PulseDO\high\PLength:=0.5,sdo_T_Rob2_StopProc;
        IDelete iMoveHome_RBT1;
        ClkStop clockWeldTime;
        nclockWeldTime{1}:=ClkRead(clockWeldTime);
        StopMove;
        ClearPath;
        StartMove;
        IF bRobSwap=FALSE THEN
            Set po36_ArcR1Error;
            MonitorweldErrorpostion.monPose1:=MonitorPosition.monPose1;
            MonitorweldErrorpostion.monPose2:=MonitorPosition.monPose2;
        ELSE
            Set po37_ArcR2Error;
            MonitorweldErrorpostion.monPose1:=MonitorPosition.monPose1;
            MonitorweldErrorpostion.monPose2:=MonitorPosition.monPose2;
        ENDIF

        pTemp:=CRobT(\TaskName:="T_ROB1"\Tool:=tWeld1\WObj:=wobjWeldLine1);
        MoveL RelTool(pTemp,0,0,-10),vTargetSpeed,z0,tWeld1\WObj:=wobjWeldLine1;
        stReact{1}:="Error_Arc_Touch";
        WaitSyncTask Wait{80},taskGroup123;

        WaitUntil stReact=["Error_Arc_Touch","Error_Arc_Touch","Error_Arc_Touch"];
        WaitSyncTask Wait{81},taskGroup123;

        WaitUntil stCommand="Error_Arc_Touch";
        stReact{1}:="";
        WaitUntil stCommand="";
        WaitSyncTask Wait{82},taskGroup123;
        Reset po14_Motion_Working;
        Set po15_Motion_Finish;
        Stop;
        ExitCycle;

    ENDPROC

    PROC rTouchErrorHandling(num Errorno)
        VAR robtarget pTemp;
        Reset soLn1Touch;
        Set po33_TouchR1Error;

        pTemp:=CRobT(\TaskName:="T_ROB1"\tool:=tWeld1\WObj:=wobjWeldLine1);
        MoveL RelTool(pTemp,0,0,-10),v200,z10,tWeld1\WObj:=wobjWeldLine1;

        stReact{1}:="Error_Arc_Touch";
        WaitSyncTask Wait{80},taskGroup123;

        WaitUntil stReact=["Error_Arc_Touch","Error_Arc_Touch","Error_Arc_Touch"];
        WaitSyncTask Wait{81},taskGroup123;

        WaitUntil stCommand="Error_Arc_Touch";
        stReact{1}:="";
        WaitUntil stCommand="";
        WaitSyncTask Wait{82},taskGroup123;

        StartMove;
        ExitCycle;

    ENDPROC

    PROC rT_ROB1check()
        VAR robtarget pTemp;
        pTemp:=CRobT(\TaskName:="T_ROB1"\Tool:=tWeld1\WObj:=wobjWeldLine1);
        IF Abs(pTemp.trans.Y)<100 AND Abs(pTemp.trans.Z)<200 THEN
            IF pTemp.trans.Y>0 THEN
                pTemp.trans.y:=130;
                MoveL pTemp,v100,fine,tWeld1\WObj:=wobjWeldLine1;
            ENDIF
            IF pTemp.trans.Y<0 THEN
                pTemp.trans.y:=-130;
                MoveL pTemp,v100,fine,tWeld1\WObj:=wobjWeldLine1;
            ENDIF
        ENDIF
    ENDPROC

    PROC rCheckWelder()
        IF (soLn1Touch=1) THEN
            Reset soLn1Touch;
            WaitTime 0.5;
        ENDIF
        WaitTime 0.5;
        WaitUntil(siLn1TouchActive=0 OR soLn1Touch=0);
        Set soLn1Touch;
        WaitUntil(siLn1TouchActive=1 AND soLn1Touch=1);
    ENDPROC
ENDMODULE
